// TIA Portal V16 export
// export: Created 2021-08-30T11:09:35.9482857Z, ExportSetting WithDefaults, DisplayName Totally Integrated Automation Portal, DisplayVersion V16 Update 3, DisplayName TIA Portal Version Control Interface, DisplayVersion V16 Update 2, DisplayName TIA Portal Openness, DisplayVersion V16 Update 3, DisplayName TIA Portal Teamcenter Gateway, DisplayVersion V16, DisplayName STEP 7 Professional, DisplayVersion V16 Update 3, DisplayName STEP 7 Safety, DisplayVersion V16, DisplayName WinCC Advanced, DisplayVersion V16 Update 3
VAR_GLOBAL   // PLC tag table "HW"
   PLC_RAW_DI AT %I0.0 : "PLC_HW_DI";
   PLC_RAW_DQ AT %Q0.0 : "PLC_HW_DQ";
   PLC_RAW_AI AT %I64.0 : "PLC_HW_AI";
   PLC_RAW_AQ AT %Q64.0 : "PLC_HW_AQ";
   ET_RAW_DI AT %I2.0 : "ET_HW_DI";
   ET_RAW_DQ AT %Q2.0 : "ET_HW_DQ";
   ET_RAW_AI AT %I68.0 : "ET_HW_AI";
   ET_RAW_AQ AT %Q68.0 : "ET_HW_AQ";
END_VAR
VAR_GLOBAL CONSTANT   // user constants
   PLC_DI : Int := 13;
   PLC_DQ : Int := 9;
   PLC_AI : Int := 1;
   PLC_AQ : Int := 1;
   ET_DI : Int := 79;
   ET_DQ : Int := 31;
   ET_AI : Int := 39;
   ET_AQ : Int := 7;
END_VAR
